FUNCTION FUN_EventTrigger : BOOL
VAR_INPUT
	IN 					: STRING(250);
	ModuleName 			: STRING;
	MessageText 		: STRING(250);
END_VAR
VAR
	
	STRINGLENGTH :			INT;
	ModuleNameOK :			BOOL;
	MessageTypeOK :			BOOL;
	MessageTextOK :			BOOL;
END_VAR

StringLength := LEN(IN);

IF StringLength <> 0 THEN
		
			STRINGLENGTH := FIND(IN,ModuleName);
			IF STRINGLENGTH > 0 THEN
				ModuleNameOK :=1;
			END_IF
			STRINGLENGTH := FIND(IN,MessageText);
			IF STRINGLENGTH > 0 THEN
				MessageTextOK :=1;
			END_IF
			
		IF ModuleNameOK AND MessageTextOK THEN
			EventTrigger2 :=1;
		END_IF
		
END_IF

END_FUNCTION

(* stored: Version 1.1.0.1, ProductVersion 3.1.4024.15
   POU FUN_EventTrigger: Id {bff79f51-18b7-4387-ae6a-4c46dfee5a14}, SpecialFunc None *)
